(* PLC project function, Dassault Systèmes ControlBuild 2024x *)
(* stored: creationDateTime 2023-10-03T11:13:46-01:00 *)

PROGRAM drill.function
  VAR_INPUT
    piece : BOOL := false;
  END_VAR
  VAR_INPUT
    emptyProd : BOOL := false;
    unitProd : BOOL := false;
    batchProd : BOOL := false;
  END_VAR
  VAR_INPUT
    acknowledgePB : BOOL := false;
  END_VAR
  VAR_INPUT
    autoMode : BOOL := false;
    manualMode : BOOL := false;
  END_VAR
  VAR_OUTPUT
    faultyState : BOOL := false;
    cycleEnd : BOOL := false;
    loadingRequest : BOOL := false;
    unloadingRequest : BOOL := false;
  END_VAR

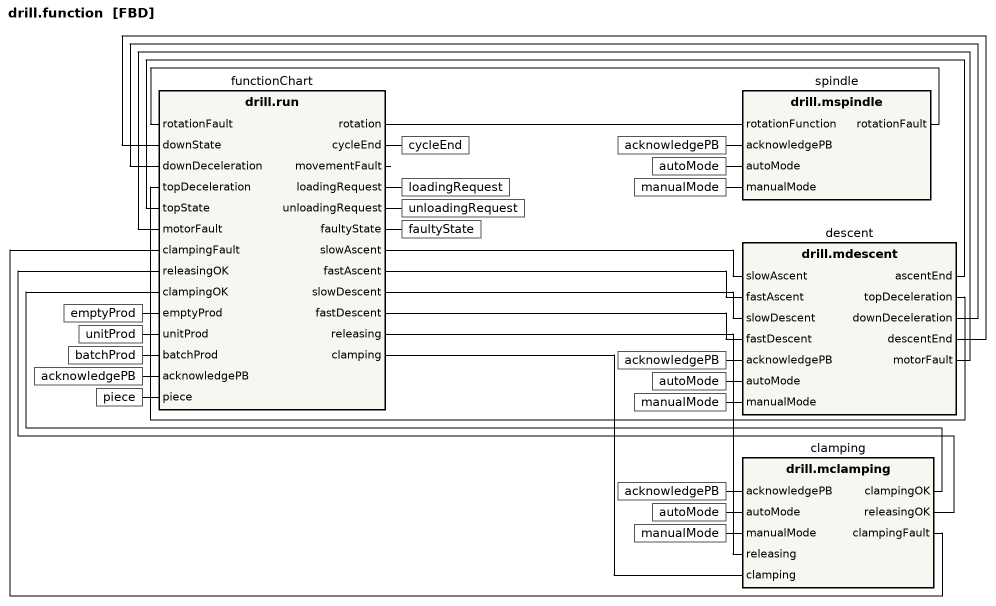
(* FBD diagram, written out as Structured Text *)
spindle(rotationFunction := functionChart.rotation, acknowledgePB := acknowledgePB, autoMode := autoMode, manualMode := manualMode);
descent(slowAscent := functionChart.slowAscent, fastAscent := functionChart.fastAscent, slowDescent := functionChart.slowDescent, fastDescent := functionChart.fastDescent, acknowledgePB := acknowledgePB, autoMode := autoMode, manualMode := manualMode);
clamping(acknowledgePB := acknowledgePB, autoMode := autoMode, manualMode := manualMode, releasing := functionChart.releasing, clamping := functionChart.clamping);
functionChart(rotationFault := spindle.rotationFault, downState := descent.descentEnd, downDeceleration := descent.downDeceleration, topDeceleration := descent.topDeceleration, topState := descent.ascentEnd, motorFault := descent.motorFault, clampingFault := clamping.clampingFault, releasingOK := clamping.releasingOK, clampingOK := clamping.clampingOK, emptyProd := emptyProd, unitProd := unitProd, batchProd := batchProd, acknowledgePB := acknowledgePB, piece := piece);
cycleEnd := functionChart.cycleEnd;
loadingRequest := functionChart.loadingRequest;
unloadingRequest := functionChart.unloadingRequest;
faultyState := functionChart.faultyState;
END_PROGRAM
